// TwinCAT 3 PLC project TEXXX_XXX
// ProgramVersion: 3.1.4024.0
// libraries:
//   Tc2_Standard, * (Beckhoff Automation GmbH)
//   Tc2_System, * (Beckhoff Automation GmbH)
//   Tc2_Utilities, * (Beckhoff Automation GmbH)
//   Tc3_Module, * (Beckhoff Automation GmbH)
// project tree:
//   DUTs/HMI/ ST_StatusBanner.TcDUT (not stored), ST_Timers.TcDUT
//   DUTs/IO/CARDS/ ST_Terminal_Info.TcDUT (not stored), ST_EL1809.TcDUT (not stored), ST_EL2809.TcDUT (not stored)
//   DUTs/MASTER/ E_MachineState.TcDUT (not stored), E_ProcessCycle.TcDUT (not stored), ST_ButtonsLamps.TcDUT (not stored), ST_HMI_IO.TcDUT (not stored), ST_MachineStatus.TcDUT (not stored), ST_MasterCTRL.TcDUT (not stored), ST_StationCMD.TcDUT (not stored), ST_StationStatus.TcDUT (not stored), ST_Puls.TcDUT (not stored), ST_StatisticsHMI.TcDUT (not stored)
//   DUTs/MASTER/log_CSV/ ST_CSVProcess.TcDUT (not stored), ST_UserLog.TcDUT (not stored), ST_CycleData.TcDUT (not stored)
//   DUTs/PDFMaker/ ST_EventsPDF.TcDUT (not stored), ST_EventsPdfConstants.TcDUT (not stored), ST_JavasCriptPDF.TcDUT (not stored), ST_PDFMaker.TcDUT (not stored)
//   DUTs/STATIONS/STATION_1/ E_Station1_State.TcDUT (not stored), ST_CycleDataStation1.TcDUT (not stored), ST_Station_1.TcDUT (not stored)
//   DUTs/STATIONS/STATION_2/ E_Station2_State.TcDUT (not stored), ST_CycleDataStation2.TcDUT (not stored), ST_Station_2.TcDUT (not stored)
//   DUTs/STATIONS/STATION_3/ E_Station3_State.TcDUT (not stored), ST_CycleDataStation3.TcDUT (not stored), ST_Station_3.TcDUT (not stored)
//   DUTs/USER_ALARMS_EVENTS/EVENTS/ ST_ActiveEvents.TcDUT (not stored), ST_EventsAssigment.TcDUT (not stored), ST_EventsAssigmentGeneral.TcDUT (not stored), ST_EventsHistory.TcDUT (not stored), ST_EVENT.TcDUT (not stored), ST_StationEvents.TcDUT (not stored)
//   DUTs/USER_ALARMS_EVENTS/ ST_UserLogHMI.TcDUT (not stored)
//   GVLs/ GVL_Constants.TcGVL (not stored), GVL_HMI.TcGVL, GVL_IO.TcGVL (not stored), GVL_Master.TcGVL (not stored), GVL_Persistent.TcGVL (not stored), GVL_Stations.TcGVL (not stored)
//   / PlcTask.TcTTO (not stored)
//   POUs/A_MASTER/ A_1_PRG_Main_Master.TcPOU, A_2_PRG_MachineCtrl.TcPOU (not stored), A_3_PRG_FaultHandling.TcPOU (not stored), A_4_PRG_MasterSystemTime.TcPOU (not stored)
//   POUs/B_STATIONS/B_1_LEAK_TEST/ B_1_1_PRG_Master_Station_1.TcPOU (not stored)
//   POUs/B_STATIONS/B_2_STATION_2/ B_2_1_PRG_Master_Station_2.TcPOU (not stored)
//   POUs/B_STATIONS/B_3_STATION_3/ B_3_1_PRG_Master_Station_3.TcPOU (not stored)
//   POUs/C_HMI/ C_1_PRG_MainHMI.TcPOU (not stored)
//   POUs/ MAIN.TcPOU (not stored)
//   POUs/Utilities/ FB_EventsManager.TcPOU (not stored), FB_PDFMaker.TcPOU, FB_UserLog.TcPOU (not stored), FB_Pulse.TcPOU (not stored), FB_TerminalInfo.TcPOU (not stored), FB_TimeControl.TcPOU (not stored), FB_WriteDataToCSV.TcPOU (not stored), PRG_Puls.TcPOU (not stored)
// real-time tasks:
//   TASK PlcTask: cycle T#10ms, priority 20, ADS port 350

// ---- DUTs/HMI/ST_Timers.TcDUT
TYPE ST_Timers :
STRUCT
	
	nStation1TimeOut				: DINT			:= 10;
	nStation2TimeOut				: DINT			:= 10;
	nStation3TimeOut				: DINT			:= 10;

END_STRUCT
END_TYPE

// ---- GVLs/GVL_HMI.TcGVL
VAR_GLOBAL
////////////////////////////////////////:	///////////////////////////////////////////////////
/////////////////////////////////////////////////////////////////////////////////////GENERIC/////////////////////////////////////////////////////////////////////////////////////

	stHMI_IO							: ST_HMI_IO;
	bQuitHMI							: BOOL;
	bShutDown							: BOOL;
	stStatusBanner						: ST_StatusBanner;
	nPopUp								: DINT;
	
	

/////////////////////////////////////////////////////////////////////////////////////SYSTEM INFO/////////////////////////////////////////////////////////////////////////////////////

	sSoftwareVersion					: STRING := ' 1.0 ';
	sSoftwareDate						: STRING := ' 10.December.2024 ';
	sTC3Version							: STRING := ' v3.1.4024.53, Runtime v3.1.4024.40 ';
	sHMIVersion							: STRING := ' TcXaeShell Version 15.0.28010.2050 D15.8 ';
	sSystemName							: STRING := ' Print & Applay Labeller ' ;
	sProjectID							: STRING := ' TE 1099 PAL' ;
	sAplication                     	: STRING := ' Print & Applay Labeller ';
	sHMIServer                			: STRING := ' ---- ';
	
	NetAmsId        	       			: T_AmsNetId := ''; // AMS-ID for com port setup 
	
/////////////////////////////////////////////////////////////////////////////////////USER LOG/////////////////////////////////////////////////////////////////////////////////////

	sUserGroupIn						: STRING;
	sUserGroupOut						: STRING;
	sUserName							: STRING;
	bUserLoggedIn						: BOOL;			
	bLogOut								: BOOL;	
	rUserLoggedIn						: R_TRIG;

/////////////////////////////////////////////////////////////////////////////////////MANUAL/////////////////////////////////////////////////////////////////////////////////////

	bEnableManual						: BOOL;
	nMainRegion							: DINT;
	bManualModeOffFlag					: BOOL;
	
END_VAR

VAR_GLOBAL PERSISTENT
	
	stTimers							: ST_Timers;

END_VAR

// ---- POUs/A_MASTER/A_1_PRG_Main_Master.TcPOU
PROGRAM A_1_PRG_Main_Master
VAR
	
	rtrigButton             				: ARRAY[1..3] OF Tc2_Standard.R_TRIG;
	ftrigButton             				: ARRAY[1..3] OF Tc2_Standard.F_TRIG; 
	
	fbStringFormatter       				: Tc2_Utilities.FB_FormatString;
	fbEventsManager							: FB_EventsManager;
	
	ntShutdown								: TC2_Utilities.NT_Shutdown;
	closeChrome 							: NT_StartProcess;
	tonUserLogOut							: TON;
	fbUserLog								: FB_UserLog;
	
	nFindAdm								: INT;
	nFindEng								: INT;
	nFindOpe								: INT;
	sUserGroupName							: STRING (255);
	sAdmGroup								: STRING (255)							:= 'Administrator';
	sEngGroup								: STRING (255)							:= 'Engineer';
	sOpeGroup								: STRING (255)							:= 'Operator';
	
	rEfficency								: STRING(510);
	
	fbSystemTime							: NT_GetTime;
	
////////////////////////////////////////////////////////////////////////////////////CSV////////////////////////////////////////////////////////////////////////////	

	//stEventsCSVProcess						:  ST_CSVProcess;
	//fbWriteDataToCSV_Events					: FB_WriteDataToCSV;
	fbPDFMaker								: FB_PDFMaker;
	stPDFMaker								: ST_PDFMaker;
	i										: DINT;
	

	
END_VAR

/////////////////////////////////////////////////////////////////////////////////////GENERAL/////////////////////////////////////////////////////////////////////////////////////
A_3_PRG_FaultHandling();
a_ACT_ButtonsLamps();
b_ACT_PDFMaker();
d_ACT_ShutdownAndQuit();
e_ACT_UserLog();
f_ACT_TerminalInfo();
g_ACT_Manual();
h_ACT_Statistics();

C_1_PRG_MainHMI();
//D_1_1_PROG_Write_Data_To_CSV();
//D_2_1_PROG_Write_Data_To_CSV();

PRG_Puls();

// System PowerUP CTRL
tonSystemPowerUP(IN:=bSystemPoweringUP, PT:=tSystemPowerUP_Time);
IF tonSystemPowerUP.Q THEN 
bSystemPoweringUP:=FALSE;
END_IF


A_4_PRG_MasterSystemTime();
/////////////////////////////////////////////////////////////////////////////////////STATIONS/////////////////////////////////////////////////////////////////////////////////////

B_1_1_PRG_Master_Station_1(CMD := CMD_Station1);
B_2_1_PRG_Master_Station_2(CMD := CMD_Station2);
B_3_1_PRG_Master_Station_3(CMD := CMD_Station3);

/////////////////////////////////////////////////////////////////////////////////////PROCESS/////////////////////////////////////////////////////////////////////////////////////

A_2_PRG_MachineCtrl();

/////////////////////////////////////////////////////////////////////////////////////EVENT LOG/////////////////////////////////////////////////////////////////////////////////////

fbEventsManager	(			//INPUTS
							bPulse 							:= stPuls.bFlash10Hz, 
							bResetFaults 					:= bResetTest, 
							stStationEvents 				:= stStationEvents,
							sSystemTime						:= sSystemTime,
							sSystemDate						:= sSystemDate,
 							stEventsAssigment				:= stEventsAssigment,
							bDataWritedInCSV				:= stPDFMaker.bDataWrited,
							
							//OUTPUTS
							astActiveEvents 				=> astActiveEvents,
							astEventsHistory				=> astEventsHistory,
							bWriteDataInCSV					=> stPDFMaker.bWriteData,
							nDataHistoryIndex				=> stPDFMaker.nDataHistoryIndex
							);



////////////////////////////////////////////////////////////////////////////////////SYSTEM DATE & TIME/////////////////////////////////////////////////////////////////////////////////////

fbSystemTime( START := stPuls.bFlash10Hz, TIMESTR => stSystemTime);
	

sSystemTime					:= 	CONCAT( STR1 := WORD_TO_STRING(stSystemTime.wHour), STR2 := CONCAT( STR1 := ':', STR2 := 
								CONCAT( STR1 := WORD_TO_STRING(stSystemTime.wMinute), STR2 := 
								CONCAT(STR1 := ':', STR2 := WORD_TO_STRING(stSystemTime.wSecond)))));
								
sSystemDate					:= 	CONCAT( STR1 := WORD_TO_STRING(stSystemTime.wDay), STR2 := 
								CONCAT(STR1 := '/', STR2 := CONCAT(STR1 := WORD_TO_STRING(stSystemTime.wMonth), STR2 := 
								CONCAT(STR1 := '/', STR2 := WORD_TO_STRING(stSystemTime.wYear)))));

ACTION a_ACT_ButtonsLamps:
//===================================================================
stButtonsLamps.bStartButtonFallingEdge 	:= ftrigButton[1].Q ;
stButtonsLamps.bStartButtonRisingEdge 	:= rtrigButton[1].Q ;
stButtonsLamps.bStopButtonFallingEdge 	:= ftrigButton[2].Q ; 
stButtonsLamps.bStopButtonRisingEdge 	:= rtrigButton[2].Q ;  
stButtonsLamps.bResetButtonFallingEdge 	:= ftrigButton[3].Q ;
stButtonsLamps.bResetButtonRisingEdge 	:= rtrigButton[3].Q ;



ftrigButton[1](CLK :=);
rtrigButton[1](CLK						:=);
ftrigButton[2](CLK						:=);
rtrigButton[2](CLK						:=);
ftrigButton[3](CLK	:=bResetTest 		);
rtrigButton[3](CLK						:=);



//GVL_IO.dw_T11_EL2809.qRESETButton_Indicator := stPuls.bFlash2Hz AND (NOT stMachineStatus.bInitialising AND NOT stMachineStatus.bAutoCycle AND NOT stMachineStatus.bManualMode AND NOT stMachineStatus.bReadyToStart) ;
//GVL_IO.dw_T11_EL2809.qStartButton_Indicator := (stPuls.bFlash2Hz AND stMachineStatus.bReadyToStart) OR (stMachineStatus.bManualMode AND stPuls.bFlash4Hz ) ;
END_ACTION

ACTION b_ACT_PDFMaker:
//EVENTS TO CSV

fbPDFMaker(					
							aDataHistory				:= astEventsHistory,
							bWriteData					:= stPDFMaker.bWriteData,
							sDate						:= stPDFMaker.sDate,
							aDataHistoryArrayLength		:= 1000,
							nDataHistoryIndex			:= stPDFMaker.nDataHistoryIndex,
							sUser						:= 'sebastian',//sUserName,
							sGroup						:= 'administrator',//sUserGroupOut,
							sMachineName				:= 'example',
							
							bDataWrited					=> stPDFMaker.bDataWrited,
							stJavasCriptPDF				=> stPDFMaker.stJavaScriptPDF
							);

(*stPDFMaker.sDate			:= 	CONCAT( STR1 := WORD_TO_STRING(stSystemTime.wDay), STR2 := 
								CONCAT(STR1 := '_', STR2 := CONCAT(STR1 := WORD_TO_STRING(stSystemTime.wMonth), STR2 := 
								CONCAT(STR1 := '_', STR2 := WORD_TO_STRING(stSystemTime.wYear)))));	*)
//CSV
(*fbWriteDataToCSV_Events( 	bWriteData					:= stEventsCSVProcess.bWriteData,
							sFileNamePath				:= stEventsCSVProcess.sFileNamePath,
							sDate						:= stEventsCSVProcess.sDate,
							aDataHistoryArrayLength		:= stEventsCSVProcess.aDataHistoryArrayLength,
							nMAX_CSV_ROWS				:= stEventsCSVProcess.nMAX_CSV_ROWS,
							nMAX_CSV_COLUMNS			:= stEventsCSVProcess.nMAX_CSV_COLUMNS,
							nDataHistoryIndex			:= stEventsCSVProcess.nDataHistoryIndex,
							
							bBusy						=> stEventsCSVProcess.bBusy,
							bError						=> stEventsCSVProcess.bError,
							nErrId						=>,
							bDataWrited					=> stEventsCSVProcess.bDataWrited,
							aDataHistory				:= astEventsHistory);
							

(*stEventsCSVProcess.sDate	:= 	CONCAT( STR1 := WORD_TO_STRING(stSystemTime.wDay), STR2 := 
								CONCAT(STR1 := '_', STR2 := CONCAT(STR1 := WORD_TO_STRING(stSystemTime.wMonth), STR2 := 
								CONCAT(STR1 := '_', STR2 := WORD_TO_STRING(stSystemTime.wYear)))));		*)				
								

stEventsCSVProcess.sFileNamePath						:= 'C:\Users\Sebastian.Ulloa\Desktop\GIT PROJECTS\TEMPLATES\TEMPLATE_VER1\CSV\EVENTS\';								
stEventsCSVProcess.aDataHistoryArrayLength				:= 200;
stEventsCSVProcess.nMAX_CSV_ROWS						:= 1000;
stEventsCSVProcess.nMAX_CSV_COLUMNS						:= 4;*)
END_ACTION

ACTION d_ACT_ShutdownAndQuit:
closeChrome(
    NetId := '',
    PathStr := 'C:\Windows\System32\mshta vbscript:Execute("CreateObject(""WScript.Shell"").Run ""powershell -c',
    DirName := 'C:\Windows\System32\WindowsPowerShell\v1.0',
    ComndLine := 'taskkill /F /IM chrome.exe /T"", 0: window.close")',
    Start := bQuitHmi,
    TmOut := DEFAULT_ADS_TIMEOUT
);
 
bQuitHmi:= FALSE;

ntShutdown(NETID := NetAmsId, DELAY := 5, START := bShutDown);
END_ACTION

ACTION e_ACT_UserLog:
sUserGroupName																:= sUserGroupIn;

nFindAdm	:= TC2_Utilities.FIND( 	STR1									:= sUserGroupName,
									STR2									:= sAdmGroup);
									
nFindEng	:= TC2_Utilities.FIND( 	STR1									:= sUserGroupName,
									STR2									:= sEngGroup);
					
nFindOpe	:= TC2_Utilities.FIND( 	STR1									:= sUserGroupName,
									STR2									:= sOpeGroup);
				
IF nFindAdm <> 0 THEN
	sUserGroupOut															:= 'Administrator';
ELSIF nFindEng <> 0 THEN
	sUserGroupOut															:= 'Engineer';
ELSIF nFindOpe <> 0 THEN
	sUserGroupOut															:= 'Operator';
ELSE sUserGroupOut															:= '';
END_IF

tonUserLogOut( IN := (sUserGroupOut <> 'Administrator' OR sUserGroupOut <> 'Engineer') AND bUserLoggedIn , PT := T#10M);

IF tonUserLogOut.Q THEN
	bLogOut 											:= TRUE;
ELSE bLogOut 											:= FALSE;
END_IF

rUserLoggedIn( CLK := bUserLoggedIn);

fbUserLog(	nNumberOfData								:= 250,
			bSaveSignal									:= rUserLoggedIn.Q, 
			sUser										:= sUserName,
			sGroup										:= sUserGroupOut,
			sDate										:= sSystemDate,
			sTime										:= sSystemTime,
			aDataOutput									:= stUserLog);
END_ACTION

ACTION f_ACT_TerminalInfo:
dw_T03_EL1809.stTerminalInfo.fbTerminalInfo( 	nTerminalState						:= dw_T03_EL1809.stTerminalInfo.nTerminal_State,
												sTerminalState						=> dw_T03_EL1809.stTerminalInfo.sTerminalInfo);
												
dw_T04_EL2809.stTerminalInfo.fbTerminalInfo(	nTerminalState						:= dw_T04_EL2809.stTerminalInfo.nTerminal_State,
												sTerminalState						=> dw_T04_EL2809.stTerminalInfo.sTerminalInfo);
END_ACTION

ACTION g_ACT_Manual:


IF stMachineStatus.bReadyToStart THEN
	bEnableManual											:= TRUE;
ELSE bEnableManual											:= FALSE;
END_IF

IF nMainRegion = 5 AND stMasterCtrl.bNoImmediateFault AND stMasterCtrl.bNoCycleStopFault
	AND NOT stMasterCtrl.bCycleStopRequest AND NOT stButtonsLamps.bStopButtonFallingEdge THEN
	stMasterCtrl.bManualModeRequest							:= TRUE;
	bManualModeOffFlag										:= FALSE;
ELSE 
	stMasterCtrl.bManualModeRequest							:= FALSE; 
	bManualModeOffFlag										:= TRUE;											
END_IF
END_ACTION

ACTION h_ACT_Statistics:
stStatisticsHMI[0].sName			:= 'TOTAL';

stStatisticsHMI[0].nGood		:= stStatisticsHMI[1].nGood + stStatisticsHMI[2].nGood + stStatisticsHMI[3].nGood;
stStatisticsHMI[0].nTotalGood	:= stStatisticsHMI[1].nTotalGood + stStatisticsHMI[2].nTotalGood + stStatisticsHMI[3].nTotalGood;
stStatisticsHMI[0].nBad			:= stStatisticsHMI[1].nBad + stStatisticsHMI[2].nBad + stStatisticsHMI[3].nBad;
stStatisticsHMI[0].nTotalBad	:= stStatisticsHMI[1].nTotalBad + stStatisticsHMI[2].nTotalBad + stStatisticsHMI[3].nTotalBad;

								

IF (( stStatisticsHMI[0].nGood + stStatisticsHMI[0].nBad) <> 0) THEN
	
	rEfficency							:= LREAL_TO_FMTSTR(in := (DINT_TO_REAL(stStatisticsHMI[0].nGood) /( DINT_TO_REAL(stStatisticsHMI[0].nGood) + DINT_TO_REAL(stStatisticsHMI[0].nBad))) * 100.0,iPrecision := 2, bRound := TRUE);
	stStatisticsHMI[0].nEfficency		:= CONCAT(STR1 := '%', STR2 := (rEfficency));

ELSE stStatisticsHMI[0].nEfficency		:= CONCAT(STR1 := '%', STR2 := (DINT_TO_STRING(0)));
	
END_IF
END_ACTION

END_PROGRAM

// ---- POUs/Utilities/FB_PDFMaker.TcPOU
FUNCTION_BLOCK FB_PDFMaker
VAR_INPUT
	
	aDataHistory			: ARRAY[0..200] OF ST_EventsHistory;
	bWriteData				: BOOL;
	aDataHistoryArrayLength	: DINT;
	nDataHistoryIndex		: DINT;
	sDate					: STRING(255);
	
	sUser					: STRING(255);
	sGroup					: STRING(255);
	sMachineName			: STRING(255);
	
	 
END_VAR
VAR_OUTPUT
	
	stJavasCriptPDF		: ST_JavasCriptPDF;
	bDataWrited			: BOOL;
	bMakePdf			: BOOL;

END_VAR
VAR
	
	rWriteData				: R_TRIG;
	i						: DINT;
	nRowIndex				: DINT;
	sPDFDate				: STRING(255);
	bWritePDF				: BOOL;
	sFileName				: STRING(255);
	tonResetData			: TON;
	TEST					: BOOL;
	
END_VAR

ACT_IO();
ACT_WriteData();

bMakePdf			:= TEST;

ACTION ACT_IO:
stJavasCriptPDF.stEventsPdfConstants.sGroup			:= sGroup;		
stJavasCriptPDF.stEventsPdfConstants.sMachineName	:= sMachineName;
stJavasCriptPDF.stEventsPdfConstants.sUser			:= sUser;
stJavasCriptPDF.stEventsPdfConstants.sFileName		:= sFileName;
END_ACTION

ACTION ACT_WriteData:
rWriteData( CLK := bWriteData);

IF rWriteData.Q THEN
	
	FOR i := 0 TO aDataHistoryArrayLength DO
				
					stJavasCriptPDF.stEventsPDF[nRowIndex + i].sEvents					:= 	aDataHistory[i].sEventTex;
					stJavasCriptPDF.stEventsPDF[nRowIndex + i].sType					:= 	aDataHistory[i].sType;
					stJavasCriptPDF.stEventsPDF[nRowIndex + i].sDate					:= 	aDataHistory[i].sDate;
					stJavasCriptPDF.stEventsPDF[nRowIndex + i].sTime					:= 	aDataHistory[i].sTime;
				
	END_FOR
	
	i													:= 0;
	
	bDataWrited											:= TRUE;
	nRowIndex											:= nRowIndex + 201;

	

END_IF

IF nDataHistoryIndex = 0 THEN
	
	bDataWrited											:= FALSE;

END_IF

IF sPDFDate <> sDate THEN
	
	bWritePDF							:= TRUE;
	sPDFDate							:= sDate;
	
END_IF

sFileName 								:= CONCAT( STR1 := 'PDF_', STR2 := sPDFDate);

tonResetData( IN := bWritePDF, PT := T#1S);

IF tonResetData.Q THEN
	
	FOR i := 0 TO 1000 DO
				
					stJavasCriptPDF.stEventsPDF[i].sDate					:= 	'';
					stJavasCriptPDF.stEventsPDF[i].sEvents					:=  '';
					stJavasCriptPDF.stEventsPDF[i].sTime					:= 	'';
					stJavasCriptPDF.stEventsPDF[i].sType					:= 	'';
				
	END_FOR
	nRowIndex 										:= 0;		
	bWritePDF										:= FALSE;
	i												:= 0;
END_IF
END_ACTION

END_FUNCTION_BLOCK
